// TIA Portal V17 export
// export: Created 2023-12-22T15:03:16.5146766Z, ExportSetting WithDefaults, DisplayName Totally Integrated Automation Portal, DisplayVersion V17, DisplayName TIA Portal Openness, DisplayVersion V17, DisplayName TIA Portal Version Control Interface, DisplayVersion V17, DisplayName STEP 7 Professional, DisplayVersion V17, DisplayName STEP 7 Safety, DisplayVersion V17, DisplayName WinCC Advanced, DisplayVersion V17
FUNCTION_BLOCK "Route_Check"   // FB3, LAD
TITLE = Проверка маршрутов для заполнения РВ
{ S7_Optimized_Access := 'TRUE' }
VERSION : 0.1
// stored: AutoNumber true, IsIECCheckEnabled false, IsRetainMemResEnabled false, MemoryReserve 100, SetENOAutomatically false, UDAEnableTagReadback false
   VAR
      ready_2_7_from_2_9 : Bool;
      ready_2_7_from_SKV13 : Bool;
      ready_2_7_from_2_6_1 : Bool;
      ready_2_7_from_2_6_2 : Bool;
      ready_2_7_q_1 : Bool;
      ready_2_7_q_2 : Bool;
      ready_2_6_from_SKV14 : Bool;
      ready_2_6_from_2_5_1 : Bool;
      ready_2_6_from_2_5_2 : Bool;
      ready_2_6_q_1 : Bool;
      ready_2_6_q_2 : Bool;
   END_VAR
BEGIN

REGION Network 1: СКВ-2
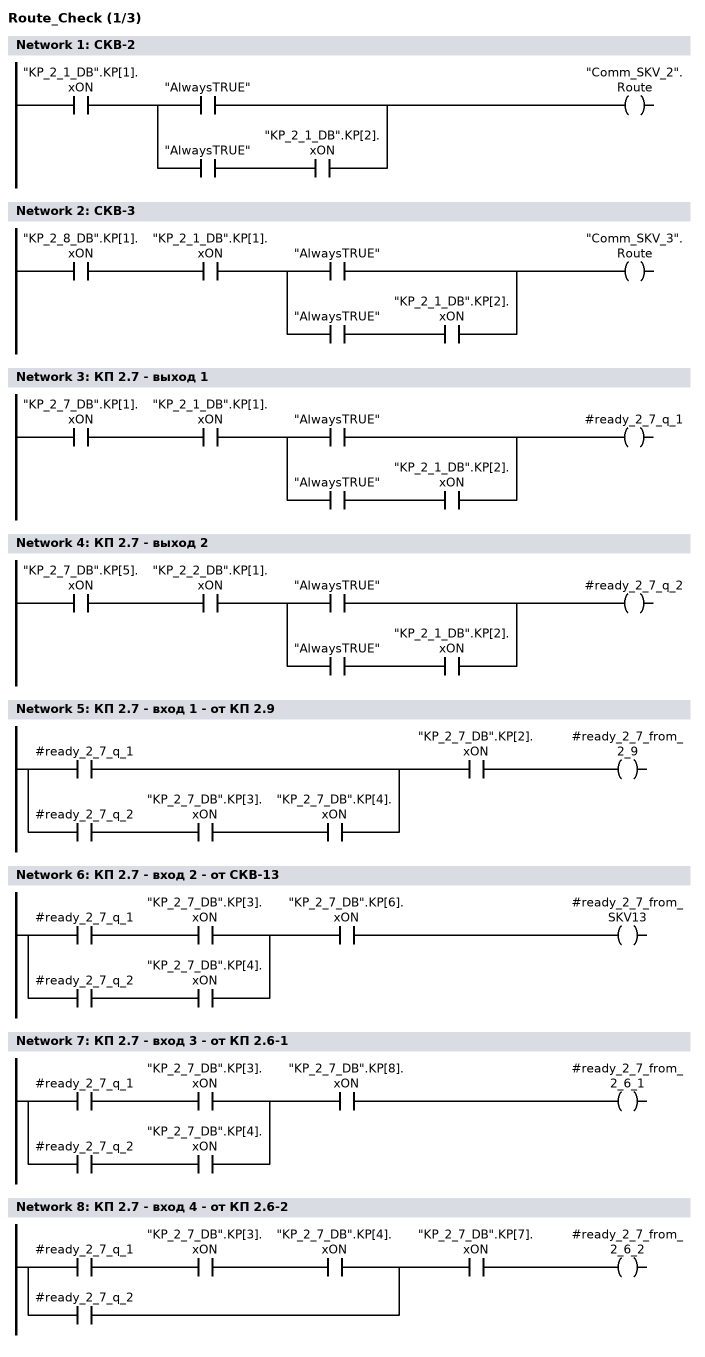
   RUNG wire#powerrail
      Contact( "KP_2_1_DB".KP[1].xON )
      wire#w1
      Contact( "AlwaysTRUE" )
      wire#w2
      Coil( "Comm_SKV_2".Route )
   END_RUNG
   RUNG wire#w1
      Contact( "AlwaysTRUE" )
      Contact( "KP_2_1_DB".KP[2].xON )
   END_RUNG wire#w2
   // the same network as SCL:
   "Comm_SKV_2".Route := "KP_2_1_DB".KP[1].xON AND ("AlwaysTRUE" OR ("AlwaysTRUE" AND "KP_2_1_DB".KP[2].xON));
END_REGION

REGION Network 2: СКВ-3
   RUNG wire#powerrail
      Contact( "KP_2_8_DB".KP[1].xON )
      Contact( "KP_2_1_DB".KP[1].xON )
      wire#w1
      Contact( "AlwaysTRUE" )
      wire#w2
      Coil( "Comm_SKV_3".Route )
   END_RUNG
   RUNG wire#w1
      Contact( "AlwaysTRUE" )
      Contact( "KP_2_1_DB".KP[2].xON )
   END_RUNG wire#w2
   // the same network as SCL:
   "Comm_SKV_3".Route := "KP_2_8_DB".KP[1].xON AND "KP_2_1_DB".KP[1].xON AND ("AlwaysTRUE" OR ("AlwaysTRUE" AND "KP_2_1_DB".KP[2].xON));
END_REGION

REGION Network 3: КП 2.7 - выход 1
   RUNG wire#powerrail
      Contact( "KP_2_7_DB".KP[1].xON )
      Contact( "KP_2_1_DB".KP[1].xON )
      wire#w1
      Contact( "AlwaysTRUE" )
      wire#w2
      Coil( #ready_2_7_q_1 )
   END_RUNG
   RUNG wire#w1
      Contact( "AlwaysTRUE" )
      Contact( "KP_2_1_DB".KP[2].xON )
   END_RUNG wire#w2
   // the same network as SCL:
   #ready_2_7_q_1 := "KP_2_7_DB".KP[1].xON AND "KP_2_1_DB".KP[1].xON AND ("AlwaysTRUE" OR ("AlwaysTRUE" AND "KP_2_1_DB".KP[2].xON));
END_REGION

REGION Network 4: КП 2.7 - выход 2
   RUNG wire#powerrail
      Contact( "KP_2_7_DB".KP[5].xON )
      Contact( "KP_2_2_DB".KP[1].xON )
      wire#w1
      Contact( "AlwaysTRUE" )
      wire#w2
      Coil( #ready_2_7_q_2 )
   END_RUNG
   RUNG wire#w1
      Contact( "AlwaysTRUE" )
      Contact( "KP_2_1_DB".KP[2].xON )
   END_RUNG wire#w2
   // the same network as SCL:
   #ready_2_7_q_2 := "KP_2_7_DB".KP[5].xON AND "KP_2_2_DB".KP[1].xON AND ("AlwaysTRUE" OR ("AlwaysTRUE" AND "KP_2_1_DB".KP[2].xON));
END_REGION

REGION Network 5: КП 2.7 - вход 1 - от КП 2.9
   RUNG wire#powerrail
      Contact( #ready_2_7_q_1 )
      wire#w1
      Contact( "KP_2_7_DB".KP[2].xON )
      Coil( #ready_2_7_from_2_9 )
   END_RUNG
   RUNG wire#powerrail
      Contact( #ready_2_7_q_2 )
      Contact( "KP_2_7_DB".KP[3].xON )
      Contact( "KP_2_7_DB".KP[4].xON )
   END_RUNG wire#w1
   // the same network as SCL:
   #ready_2_7_from_2_9 := (#ready_2_7_q_1 OR (#ready_2_7_q_2 AND "KP_2_7_DB".KP[3].xON AND "KP_2_7_DB".KP[4].xON)) AND "KP_2_7_DB".KP[2].xON;
END_REGION

REGION Network 6: КП 2.7 - вход 2 - от СКВ-13
   RUNG wire#powerrail
      Contact( #ready_2_7_q_1 )
      Contact( "KP_2_7_DB".KP[3].xON )
      wire#w1
      Contact( "KP_2_7_DB".KP[6].xON )
      Coil( #ready_2_7_from_SKV13 )
   END_RUNG
   RUNG wire#powerrail
      Contact( #ready_2_7_q_2 )
      Contact( "KP_2_7_DB".KP[4].xON )
   END_RUNG wire#w1
   // the same network as SCL:
   #ready_2_7_from_SKV13 := ((#ready_2_7_q_1 AND "KP_2_7_DB".KP[3].xON) OR (#ready_2_7_q_2 AND "KP_2_7_DB".KP[4].xON)) AND "KP_2_7_DB".KP[6].xON;
END_REGION

REGION Network 7: КП 2.7 - вход 3 - от КП 2.6-1
   RUNG wire#powerrail
      Contact( #ready_2_7_q_1 )
      Contact( "KP_2_7_DB".KP[3].xON )
      wire#w1
      Contact( "KP_2_7_DB".KP[8].xON )
      Coil( #ready_2_7_from_2_6_1 )
   END_RUNG
   RUNG wire#powerrail
      Contact( #ready_2_7_q_2 )
      Contact( "KP_2_7_DB".KP[4].xON )
   END_RUNG wire#w1
   // the same network as SCL:
   #ready_2_7_from_2_6_1 := ((#ready_2_7_q_1 AND "KP_2_7_DB".KP[3].xON) OR (#ready_2_7_q_2 AND "KP_2_7_DB".KP[4].xON)) AND "KP_2_7_DB".KP[8].xON;
END_REGION

REGION Network 8: КП 2.7 - вход 4 - от КП 2.6-2
   RUNG wire#powerrail
      Contact( #ready_2_7_q_1 )
      Contact( "KP_2_7_DB".KP[3].xON )
      Contact( "KP_2_7_DB".KP[4].xON )
      wire#w1
      Contact( "KP_2_7_DB".KP[7].xON )
      Coil( #ready_2_7_from_2_6_2 )
   END_RUNG
   RUNG wire#powerrail
      Contact( #ready_2_7_q_2 )
   END_RUNG wire#w1
   // the same network as SCL:
   #ready_2_7_from_2_6_2 := ((#ready_2_7_q_1 AND "KP_2_7_DB".KP[3].xON AND "KP_2_7_DB".KP[4].xON) OR #ready_2_7_q_2) AND "KP_2_7_DB".KP[7].xON;
END_REGION

REGION Network 9: СКВ-23
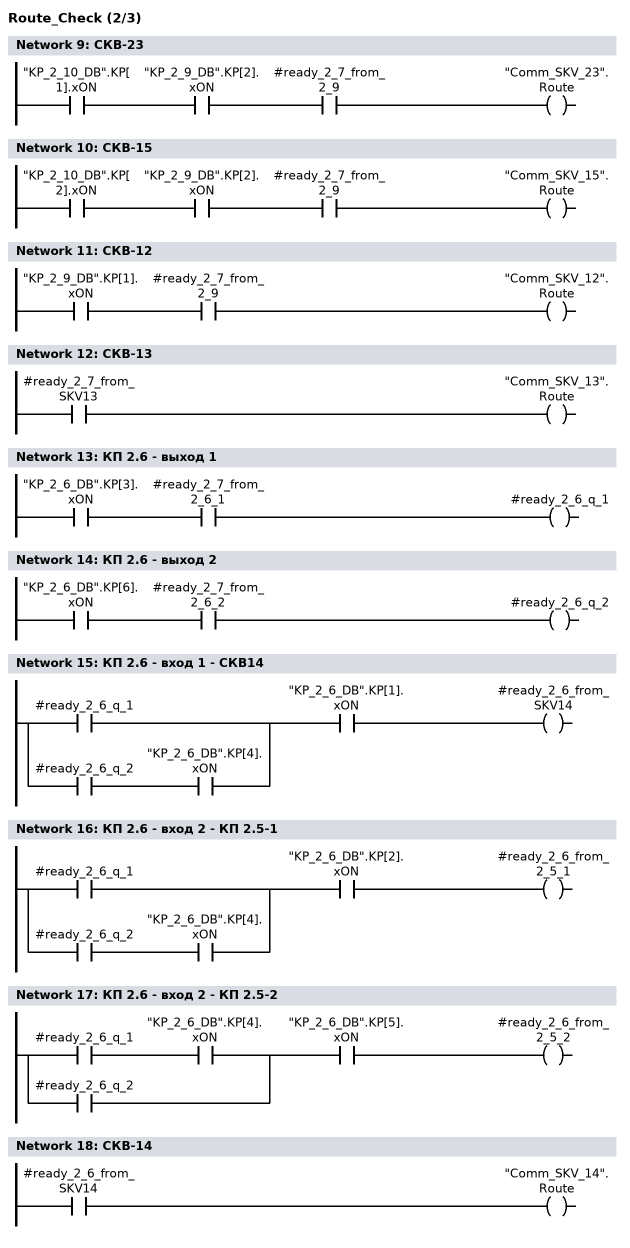
   RUNG wire#powerrail
      Contact( "KP_2_10_DB".KP[1].xON )
      Contact( "KP_2_9_DB".KP[2].xON )
      Contact( #ready_2_7_from_2_9 )
      Coil( "Comm_SKV_23".Route )
   END_RUNG
   // the same network as SCL:
   "Comm_SKV_23".Route := "KP_2_10_DB".KP[1].xON AND "KP_2_9_DB".KP[2].xON AND #ready_2_7_from_2_9;
END_REGION

REGION Network 10: СКВ-15
   RUNG wire#powerrail
      Contact( "KP_2_10_DB".KP[2].xON )
      Contact( "KP_2_9_DB".KP[2].xON )
      Contact( #ready_2_7_from_2_9 )
      Coil( "Comm_SKV_15".Route )
   END_RUNG
   // the same network as SCL:
   "Comm_SKV_15".Route := "KP_2_10_DB".KP[2].xON AND "KP_2_9_DB".KP[2].xON AND #ready_2_7_from_2_9;
END_REGION

REGION Network 11: СКВ-12
   RUNG wire#powerrail
      Contact( "KP_2_9_DB".KP[1].xON )
      Contact( #ready_2_7_from_2_9 )
      Coil( "Comm_SKV_12".Route )
   END_RUNG
   // the same network as SCL:
   "Comm_SKV_12".Route := "KP_2_9_DB".KP[1].xON AND #ready_2_7_from_2_9;
END_REGION

REGION Network 12: СКВ-13
   RUNG wire#powerrail
      Contact( #ready_2_7_from_SKV13 )
      Coil( "Comm_SKV_13".Route )
   END_RUNG
   // the same network as SCL:
   "Comm_SKV_13".Route := #ready_2_7_from_SKV13;
END_REGION

REGION Network 13: КП 2.6 - выход 1
   RUNG wire#powerrail
      Contact( "KP_2_6_DB".KP[3].xON )
      Contact( #ready_2_7_from_2_6_1 )
      Coil( #ready_2_6_q_1 )
   END_RUNG
   // the same network as SCL:
   #ready_2_6_q_1 := "KP_2_6_DB".KP[3].xON AND #ready_2_7_from_2_6_1;
END_REGION

REGION Network 14: КП 2.6 - выход 2
   RUNG wire#powerrail
      Contact( "KP_2_6_DB".KP[6].xON )
      Contact( #ready_2_7_from_2_6_2 )
      Coil( #ready_2_6_q_2 )
   END_RUNG
   // the same network as SCL:
   #ready_2_6_q_2 := "KP_2_6_DB".KP[6].xON AND #ready_2_7_from_2_6_2;
END_REGION

REGION Network 15: КП 2.6 - вход 1 - СКВ14
   RUNG wire#powerrail
      Contact( #ready_2_6_q_1 )
      wire#w1
      Contact( "KP_2_6_DB".KP[1].xON )
      Coil( #ready_2_6_from_SKV14 )
   END_RUNG
   RUNG wire#powerrail
      Contact( #ready_2_6_q_2 )
      Contact( "KP_2_6_DB".KP[4].xON )
   END_RUNG wire#w1
   // the same network as SCL:
   #ready_2_6_from_SKV14 := (#ready_2_6_q_1 OR (#ready_2_6_q_2 AND "KP_2_6_DB".KP[4].xON)) AND "KP_2_6_DB".KP[1].xON;
END_REGION

REGION Network 16: КП 2.6 - вход 2 - КП 2.5-1
   RUNG wire#powerrail
      Contact( #ready_2_6_q_1 )
      wire#w1
      Contact( "KP_2_6_DB".KP[2].xON )
      Coil( #ready_2_6_from_2_5_1 )
   END_RUNG
   RUNG wire#powerrail
      Contact( #ready_2_6_q_2 )
      Contact( "KP_2_6_DB".KP[4].xON )
   END_RUNG wire#w1
   // the same network as SCL:
   #ready_2_6_from_2_5_1 := (#ready_2_6_q_1 OR (#ready_2_6_q_2 AND "KP_2_6_DB".KP[4].xON)) AND "KP_2_6_DB".KP[2].xON;
END_REGION

REGION Network 17: КП 2.6 - вход 2 - КП 2.5-2
   RUNG wire#powerrail
      Contact( #ready_2_6_q_1 )
      Contact( "KP_2_6_DB".KP[4].xON )
      wire#w1
      Contact( "KP_2_6_DB".KP[5].xON )
      Coil( #ready_2_6_from_2_5_2 )
   END_RUNG
   RUNG wire#powerrail
      Contact( #ready_2_6_q_2 )
   END_RUNG wire#w1
   // the same network as SCL:
   #ready_2_6_from_2_5_2 := ((#ready_2_6_q_1 AND "KP_2_6_DB".KP[4].xON) OR #ready_2_6_q_2) AND "KP_2_6_DB".KP[5].xON;
END_REGION

REGION Network 18: СКВ-14
   RUNG wire#powerrail
      Contact( #ready_2_6_from_SKV14 )
      Coil( "Comm_SKV_14".Route )
   END_RUNG
   // the same network as SCL:
   "Comm_SKV_14".Route := #ready_2_6_from_SKV14;
END_REGION

REGION Network 19: СКВ-1
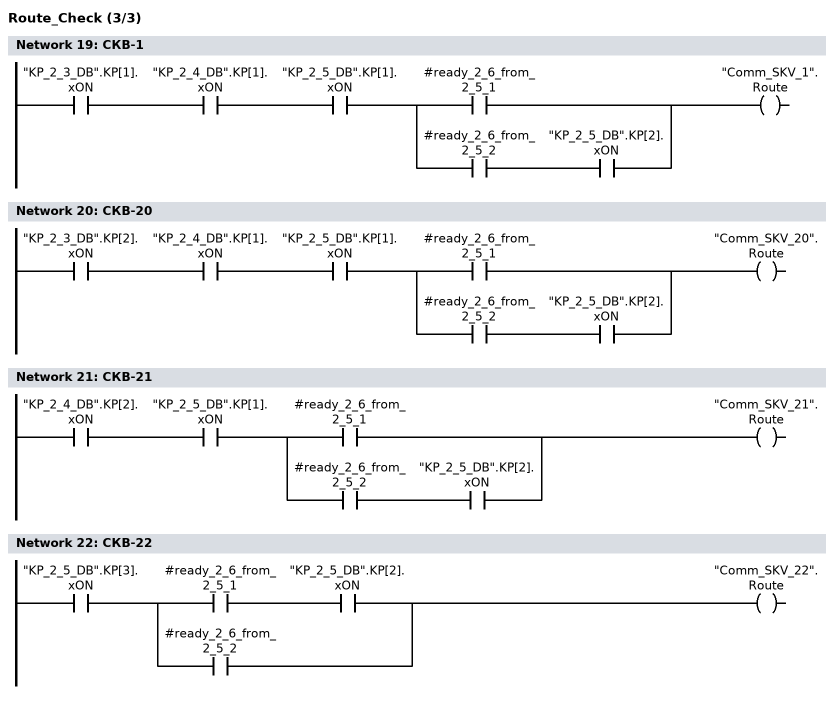
   RUNG wire#powerrail
      Contact( "KP_2_3_DB".KP[1].xON )
      Contact( "KP_2_4_DB".KP[1].xON )
      Contact( "KP_2_5_DB".KP[1].xON )
      wire#w1
      Contact( #ready_2_6_from_2_5_1 )
      wire#w2
      Coil( "Comm_SKV_1".Route )
   END_RUNG
   RUNG wire#w1
      Contact( #ready_2_6_from_2_5_2 )
      Contact( "KP_2_5_DB".KP[2].xON )
   END_RUNG wire#w2
   // the same network as SCL:
   "Comm_SKV_1".Route := "KP_2_3_DB".KP[1].xON AND "KP_2_4_DB".KP[1].xON AND "KP_2_5_DB".KP[1].xON AND (#ready_2_6_from_2_5_1 OR (#ready_2_6_from_2_5_2 AND "KP_2_5_DB".KP[2].xON));
END_REGION

REGION Network 20: СКВ-20
   RUNG wire#powerrail
      Contact( "KP_2_3_DB".KP[2].xON )
      Contact( "KP_2_4_DB".KP[1].xON )
      Contact( "KP_2_5_DB".KP[1].xON )
      wire#w1
      Contact( #ready_2_6_from_2_5_1 )
      wire#w2
      Coil( "Comm_SKV_20".Route )
   END_RUNG
   RUNG wire#w1
      Contact( #ready_2_6_from_2_5_2 )
      Contact( "KP_2_5_DB".KP[2].xON )
   END_RUNG wire#w2
   // the same network as SCL:
   "Comm_SKV_20".Route := "KP_2_3_DB".KP[2].xON AND "KP_2_4_DB".KP[1].xON AND "KP_2_5_DB".KP[1].xON AND (#ready_2_6_from_2_5_1 OR (#ready_2_6_from_2_5_2 AND "KP_2_5_DB".KP[2].xON));
END_REGION

REGION Network 21: СКВ-21
   RUNG wire#powerrail
      Contact( "KP_2_4_DB".KP[2].xON )
      Contact( "KP_2_5_DB".KP[1].xON )
      wire#w1
      Contact( #ready_2_6_from_2_5_1 )
      wire#w2
      Coil( "Comm_SKV_21".Route )
   END_RUNG
   RUNG wire#w1
      Contact( #ready_2_6_from_2_5_2 )
      Contact( "KP_2_5_DB".KP[2].xON )
   END_RUNG wire#w2
   // the same network as SCL:
   "Comm_SKV_21".Route := "KP_2_4_DB".KP[2].xON AND "KP_2_5_DB".KP[1].xON AND (#ready_2_6_from_2_5_1 OR (#ready_2_6_from_2_5_2 AND "KP_2_5_DB".KP[2].xON));
END_REGION

REGION Network 22: СКВ-22
   RUNG wire#powerrail
      Contact( "KP_2_5_DB".KP[3].xON )
      wire#w1
      Contact( #ready_2_6_from_2_5_1 )
      Contact( "KP_2_5_DB".KP[2].xON )
      wire#w2
      Coil( "Comm_SKV_22".Route )
   END_RUNG
   RUNG wire#w1
      Contact( #ready_2_6_from_2_5_2 )
   END_RUNG wire#w2
   // the same network as SCL:
   "Comm_SKV_22".Route := "KP_2_5_DB".KP[3].xON AND ((#ready_2_6_from_2_5_1 AND "KP_2_5_DB".KP[2].xON) OR #ready_2_6_from_2_5_2);
END_REGION
END_FUNCTION_BLOCK
